Staubli VAL3: sendJState.pgx

public program sendJState()
  local num l_nRetVal
begin
  call sendData(siTcpIpFbk,rosJointMsg.prefix.nData,nDataOut)
  call sendData(siTcpIpFbk,rosJointMsg.header.nData,nDataOut)
  call sendData(siTcpIpFbk,rosJointMsg.body.nData,nDataOut)
end
